{attribute 'linkalways'} 
{attribute 'no_explicit_call' := 'This FB is a CLASS and must be accessed using methods or properties'}
{attribute 'enable_dynamic_creation'}
FUNCTION_BLOCK _ETcVnRectangleIntersection EXTENDS EnumDatatypeBase
VAR
	localData : ETcVnRectangleIntersection;
	activeData : REFERENCE TO ETcVnRectangleIntersection;
	enumBaseDatatype : _DINT(localData);
END_VAR

METHOD PRIVATE AddLocalEnumeration
VAR_INPUT
	Enumeration : T_MAXSTRING;
	Value : ETcVnRectangleIntersection;
END_VAR
AddEnumeration(Enumeration, Value);
END_METHOD

PROPERTY PUBLIC Address : PVOID
GET
Address := ADR(activeData);
END_GET
END_PROPERTY

METHOD PUBLIC ClearReference
VAR_INPUT
END_VAR
activeData REF= localData;
SetBaseDatatypeReference();
END_METHOD

METHOD PUBLIC Clone : I_Datatype
VAR
    pClone : POINTER TO _ETcVnRectangleIntersection;
END_VAR
pClone := __NEW(_ETcVnRectangleIntersection(InitialValue := Value));
Clone := pClone^;
END_METHOD

METHOD FB_init : BOOL
VAR_INPUT
	bInitRetains : BOOL; // if TRUE, the retain variables are initialized (warm start / cold start)
	bInCopyCode : BOOL;  // if TRUE, the instance afterwards gets moved into the copy code (online change)
	InitialValue : ETcVnRectangleIntersection;
END_VAR
localData := InitialValue;
AddBaseDatatype(enumBaseDatatype);
ClearReference();

AddLocalEnumeration('TCVN_RI_NONE', ETcVnRectangleIntersection.TCVN_RI_NONE);
AddLocalEnumeration('TCVN_RI_PARTIAL', ETcVnRectangleIntersection.TCVN_RI_PARTIAL);
AddLocalEnumeration('TCVN_RI_FULL', ETcVnRectangleIntersection.TCVN_RI_FULL);
END_METHOD

PROPERTY PUBLIC Identifier : T_MAXSTRING
GET
Identifier := 'ETcVnRectangleIntersection';
END_GET
END_PROPERTY

METHOD IsEnumeratorValueEqual : BOOL
VAR_INPUT
	Enumerator : I_KeyValueForwardEnumerator;
END_VAR
VAR
	storedValue : ETcVnRectangleIntersection;
END_VAR
IF NOT Enumerator.TryGet(storedValue) THEN
	RETURN;
END_IF

IsEnumeratorValueEqual := storedValue = activeData;
END_METHOD

METHOD PUBLIC MakeReferenceTo
VAR_INPUT
	ReferenceTarget : REFERENCE TO ETcVnRectangleIntersection;
END_VAR
activeData REF= ReferenceTarget;
SetBaseDatatypeReference();
END_METHOD

METHOD PROTECTED SetBaseDatatypeReference
VAR_INPUT
END_VAR
enumBaseDatatype.MakeReferenceTo(activeData);
END_METHOD

PROPERTY PUBLIC Size : UDINT
GET
Size := SIZEOF(activeData);
END_GET
END_PROPERTY

METHOD TryMakeReferenceTo : BOOL
VAR_INPUT
	Target : I_Datatype;
END_VAR
VAR
	targetAsEnum : I_EnumDatatype;
	pTargetData : POINTER TO ETcVnRectangleIntersection;
END_VAR
IF NOT Target.TryResolveAsEnumDatatype(targetAsEnum) THEN
	RETURN;
END_IF

IF targetAsEnum.Identifier <> Identifier THEN
	RETURN;
END_IF

pTargetData := Target.Address;
activeData REF= pTargetData^;
SetBaseDatatypeReference();
TryMakeReferenceTo := TRUE;
END_METHOD

PROPERTY PUBLIC Value : ETcVnRectangleIntersection
GET
Value := activeData;
END_GET
SET
activeData := Value;
END_SET
END_PROPERTY

END_FUNCTION_BLOCK

(* stored: Version 1.1.0.1, ProductVersion 3.1.4024.12
   POU _ETcVnRectangleIntersection: Id {f685e4cf-73da-0f60-34df-888d73166cca}, SpecialFunc None
   Folder Constructor: Id {012c82cb-2da0-000e-02e3-ab3d88ae6286}
   Folder Private: Id {9f960bd6-1b6b-0df5-1859-4343d173f9f7}
   Folder Protected: Id {af9aed87-b539-02cf-2cf8-fd332c909b1c}
   Method AddLocalEnumeration: Id {2a9acf83-61c8-0434-2870-0d752fe5c8d2}
   Property Address: Id {6e413944-48ef-04f9-0726-2bf03fd97d66}
   Get Get: Id {75df9ff7-2d1d-02fc-2d38-b83ed89a34b4}
   Method ClearReference: Id {29b3860f-60d6-0a92-3cfb-3792c5b3d168}
   Method Clone: Id {7da9f00d-9a65-01c7-3fe0-bc441af89191}
   Method FB_init: Id {4c6f8307-ae3e-0f22-37f4-0a49d9e9ea7e}
   Property Identifier: Id {667a2cf4-6751-0df4-3456-afe11efe0d34}
   Get Get: Id {9e4fc3c9-8d29-088a-0f3e-11aa71620f7a}
   Method IsEnumeratorValueEqual: Id {4037d5e4-b8c5-0199-341e-38d3dd86c334}
   Method MakeReferenceTo: Id {6f879c8a-ba8b-0ead-12fa-4f005c6b5472}
   Method SetBaseDatatypeReference: Id {289ff085-53af-0da9-3c46-0f8db7227433}
   Property Size: Id {2e1ad109-4988-03bf-1b42-35d664880d6e}
   Get Get: Id {77c8c3f3-0315-0975-39bf-5b19e3f149cb}
   Method TryMakeReferenceTo: Id {723c4607-63d0-07fd-1a7d-c991a20526aa}
   Property Value: Id {ab343ea5-b4bd-0f61-0930-84ce8d94ebd0}
   Get Get: Id {7e76988f-5e70-04dd-1d8b-8e8717301a76}
   Set Set: Id {3f07b056-eb3f-0d93-3ace-051d02dfc4d4} *)
